PROGRAM MAIN
VAR
END_VAR

END_PROGRAM

(* stored: Version 1.1.0.1
   POU MAIN: Id {8900fb58-4648-406f-a2d8-8c1591efaa72} *)
